{attribute 'qualified_only'}
{attribute 'strict'}
TYPE MoverDirection_e :
(
	Farward,
	Reverse
);
END_TYPE

(* stored: Version 1.1.0.1, ProductVersion 3.1.4024.12
   EnumerationTextList MoverDirection_e: Id {cca35731-16ce-4880-a6b9-3a50e78a3463} *)
